RESOURCE_TYPE FakePacemakerTop
  (* Standard: 61499-2 *)
  (* Version 0.1, 2017-00-06, hpea485, UOA *)
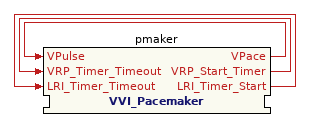
  FBS
    pmaker : VVI_Pacemaker;
  END_FBS
  EVENT_CONNECTIONS
    pmaker.VPace TO pmaker.VPulse;
    pmaker.VRP_Start_Timer TO pmaker.VRP_Timer_Timeout;
    pmaker.LRI_Timer_Start TO pmaker.LRI_Timer_Timeout;
  END_CONNECTIONS
END_RESOURCE_TYPE
